PROGRAM P_BACnet_Motion
VAR
	dwMotion	: DWORD;	//pseudo-array for storing motion (BV) information
	rMotion		: REAL;		//dwMotion converted to REAL
END_VAR

//read motion sensor's flags and combine them into DWORD (pseudo-array)
dwMotion.0 := GVL_IO.arrStreetLamps[1].bMotionFlag;
dwMotion.1 := GVL_IO.arrStreetLamps[2].bMotionFlag;
dwMotion.2 := GVL_IO.arrStreetLamps[3].bMotionFlag;
dwMotion.3 := GVL_IO.arrStreetLamps[4].bMotionFlag;
dwMotion.4 := GVL_IO.arrStreetLamps[5].bMotionFlag;
dwMotion.5 := GVL_IO.arrStreetLamps[6].bMotionFlag;
dwMotion.6 := GVL_IO.arrStreetLamps[7].bMotionFlag;
dwMotion.7 := GVL_IO.arrStreetLamps[8].bMotionFlag;
dwMotion.8 := GVL_IO.arrStreetLamps[9].bMotionFlag;
dwMotion.9 := GVL_IO.arrStreetLamps[10].bMotionFlag;

//type conversion from DWORD to REAL
rMotion := DWORD_TO_REAL(dwMotion);

//write rMotion to BACnet obcject present value
//thereby keep BACnet object instance alive
fbBACnet_AV_SL_Motion(Device := Device, bEnablePV := TRUE, bNullPV := FALSE, fPV := rMotion);

END_PROGRAM

(* stored: Version 1.1.0.1, ProductVersion 3.1.4024.5
   POU P_BACnet_Motion: Id {37b66c7f-db2a-4d9c-abd1-8561dc193161}, SpecialFunc None *)
